(* PLC project Unnamed, Unknown Unnamed 1 *)
(* stored: creationDateTime 2022-02-28T09:43:47, modificationDateTime 2022-03-30T01:32:22 *)

PROGRAM program0
  VAR
    LocalVar0 : BOOL;
    LocalVar1 : BOOL;
    LocalVar2 : BOOL;
    LocalVar3 : BOOL;
    TON0 : TON;
    TON1 : TON;
    TON2 : TON;
  END_VAR

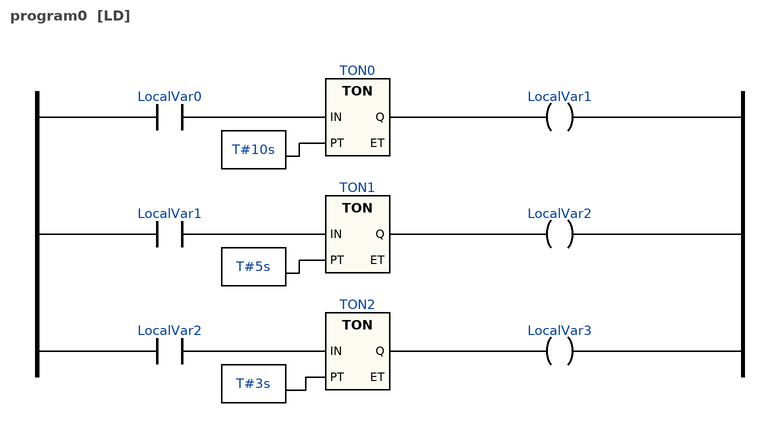
(* LD diagram, written out as Structured Text *)
TON0(IN := LocalVar0, PT := T#10s);
LocalVar1 := TON0.Q;
TON1(IN := LocalVar1, PT := T#5s);
LocalVar2 := TON1.Q;
TON2(IN := LocalVar2, PT := T#3s);
LocalVar3 := TON2.Q;
END_PROGRAM

CONFIGURATION Config0
  RESOURCE Res0 ON PLC
    TASK task0(INTERVAL := T#20ms, PRIORITY := 0);
    PROGRAM instance0 WITH task0 : program0;
  END_RESOURCE
END_CONFIGURATION
